Fanuc KAREL source: kc00033.KL

-- PROVISIONAL review KL for V770-1; original PC SHA256 d51eac3ca72ce77636a6e5b249042807e71a93be9c7493c9c2447d9f759de82f
-- Incomplete behavior may be omitted. Consult companion uncertainty JSON. Do not deploy.
PROGRAM KC00033
%NOLOCKGROUP
BEGIN
  -- UNRESOLVED_PC offsets 5-32; opcodes 27,22,1C,22,22,76
  -- UNRESOLVED_PC offsets 37-41; opcodes 7F
END KC00033
